(* Logix 5000 project; controller TestController vendor 1 type 14 code 166 rev 32.11; software revision 32.02 *)
// This is a test project

TASK Continuous (continuous, watchdog 500 ms) : MainProgram   // Test continuous task
TASK Event (event, rate 11 ms, priority 10, watchdog 500 ms)   // TestEvent Task
TASK Periodic (periodic, rate 10 ms, priority 10, watchdog 500 ms)

MODULES
   Local : vendor 1 type 14 code 166 (ICP 0, rev 32.11)
      RakIO : 1756-EN2T (Ethernet 10.10.10.10, rev 11.1, Output RPI 10 ms)   // This is a test EN2T module
         Module1 : 1756-IB16 (ICP 1, rev 3.1)
         Mod5 : 1756-IB16 (ICP 3, rev 3.1)
              RakIO:3:I.Data.0   // IO Description
         IF8 : 1756-IF8 (ICP 2, rev 1.1, Input RPI 100 ms)   // Ths is a test IF8
      FlexIO : 5094-AEN2TR (Ethernet 10.11.12.13, rev 4.1)
         Flex_Mod_1 : 5094-IF8 (5094 1, rev 2.1, StandardDataDriven RPI 100 ms)
         Flex_Mod_3 : 5094-IB16 (5094 3, rev 2.1, StandardDataDriven RPI 5 ms)
         Flex_Mod_2 : 5094-OB16 (5094 2, rev 2.1, StandardDataDriven RPI 5 ms)
      NewFlex : 5094-AEN2TR (Ethernet 1.2.4.0, rev 4.1)
END_MODULES

TYPE AlarmType :   // This is a test alarm type
STRUCT
   DigitalMember : CAM;   // Test digital member
END_STRUCT
END_TYPE

TYPE BoolTest :   // This is a test
STRUCT
   Member01 : BOOL;
   Member02 : BOOL;
   Member04 : BOOL;
   Member05 : BOOL;
END_STRUCT
END_TYPE

TYPE ModuleType :   // This is a test of a type that references Module-Defined types
STRUCT
   AIChannel : CHANNEL_AI:O:0;   // This is a test
END_STRUCT
END_TYPE

TYPE MyStringType :   // This is a test string type
STRUCT
   LEN : DINT;
   DATA : SINT[100];
END_STRUCT
END_TYPE

ADD_ON_INSTRUCTION aoi_Test   (* revision 1.0 *)
// Test AOI
VAR_INPUT
   InputTest : BOOL; {visible}
   OutputTest : DINT; {access Read Only, visible}
END_VAR
VAR_IN_OUT
   InOutTest : SimpleType; {required}
END_VAR
VAR_INPUT
   Config : INT; {access None, required}
   Test : BOOL; {access None}
END_VAR
VAR_IN_OUT
   Timers : REAL[5]; {required}
END_VAR
VAR
   LocalBool : BOOL; {access None}
END_VAR

ROUTINE Logic   (* ladder *)
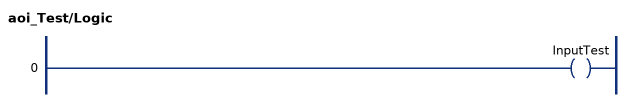
   0: OTE(InputTest);
END_ROUTINE
END_ADD_ON_INSTRUCTION

VAR_GLOBAL   (* controller tags *)
   _Test : DINT;
   aoiTestInstance : aoi_Test;
   RealArray : REAL[5];
   SimpleArray : DINT[10]; {access Read Only}   // This is a test
   SimpleBool : BOOL; {access None}
   SimpleDint : DINT := 1234567; {access None}
   SimpleInt : INT := 20; {access None}
   SimpleLint : LINT := 20; {access None}
   SimpleReal : REAL; {access None}
   SimpleSint : SINT := 16#14; {access None}
        .0   // This is a test
   TagParameter : SimpleType; {access None}
   TestAlarmTag : ALARM; {access None}   // Alarm
   TestAnalogAlarm : ALARM_ANALOG;
   TestArrayTag : ArrayType; {access Read Only}   // Base
   TestComplexTag : ComplexType; {access None}   // Base
   TestDigitalAlarm : ALARM_DIGITAL;
   TestSimpleTag : SimpleType := (IntMember := 14, DintMember := '$00$00$00$01'); {access Read Only}   // Override
   TestStringTag : MyStringType; {access None}   // String
        .DATA   // Data
   TestTimer : TIMER := (PRE := 1000); {access None}   // Test Timer
   TimerArray : TIMER[5];   // Base Timer
        [1].PRE   // PRE 1
        [1]   // Index 1
END_VAR

PROGRAM FolderProgram
END_PROGRAM

PROGRAM MainProgram   (* main routine Main *)
VAR
   Step_000 : SFC_STEP := (Status := 16#0020_0000, PauseTimer := 1);
   Tran_000 : BOOL;
END_VAR

ROUTINE FBD   (* function block diagram *)
   SHEET 1
END_ROUTINE

ROUTINE Main   (* ladder *)
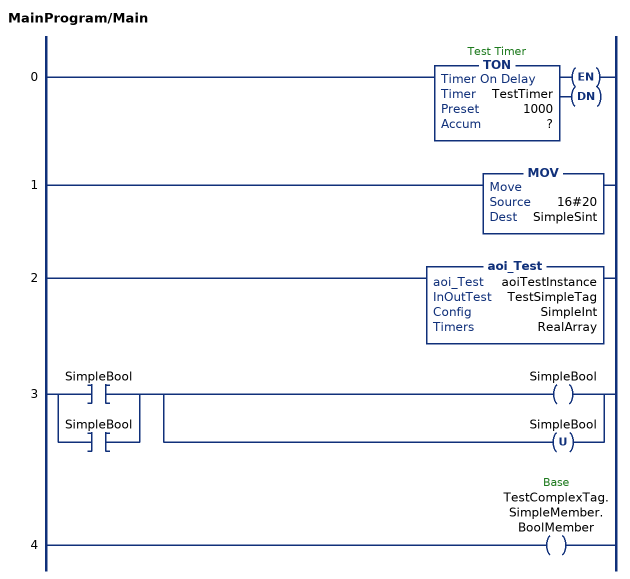
   0: TON(TestTimer,?,?);
   1: MOV(16#20,SimpleSint);
   2: aoi_Test(aoiTestInstance,TestSimpleTag,SimpleInt,RealArray);
   3: [XIC(SimpleBool) ,XIC(SimpleBool) ][OTE(SimpleBool) ,OTU(SimpleBool) ];
   4: OTE(TestComplexTag.SimpleMember.BoolMember);
END_ROUTINE

ROUTINE SFCRoutine   (* sequential function chart *)
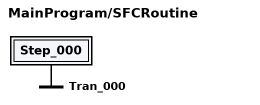
   INITIAL_STEP Step_000:
   END_STEP
   TRANSITION Tran_000 FROM Step_000 TO ()
      := 
   END_TRANSITION
END_ROUTINE

ROUTINE ST   (* structured text *)
   
END_ROUTINE
END_PROGRAM
